Omron CX-Programmer project NewProject (CX-Programmer 9.61)

# PLC NewPLC1: CJ1M CPU21
I/O table (CPU CJ1M-CPU21): rack 0 slot 0 CJ1W-ID211; rack 0 slot 1 CJ1W-OC211; rack 0 slot 2 CJ1W-MAD42

## Global symbols (name address type ; comment)
0.01 BOOL  ; START
1.00 BOOL  ; ON
1.01 BOOL  ; GERAK1
1.02 BOOL  ; GERAK2
1.03 BOOL  ; GERAK3
1.04 BOOL  ; PENGISIAN
2005 CHANNEL  ; LEVEL
T0004 BOOL  ; COUNTER

## Program NewProgram1 (cyclic task 0)

### Section Section1

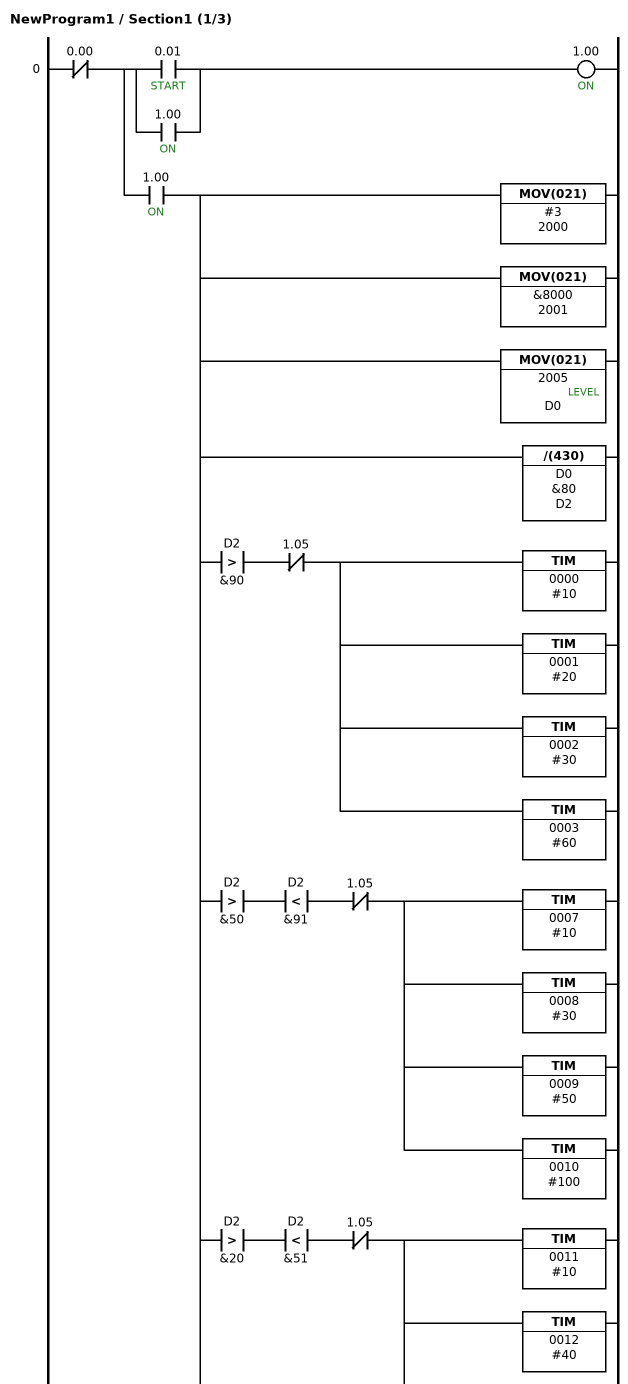

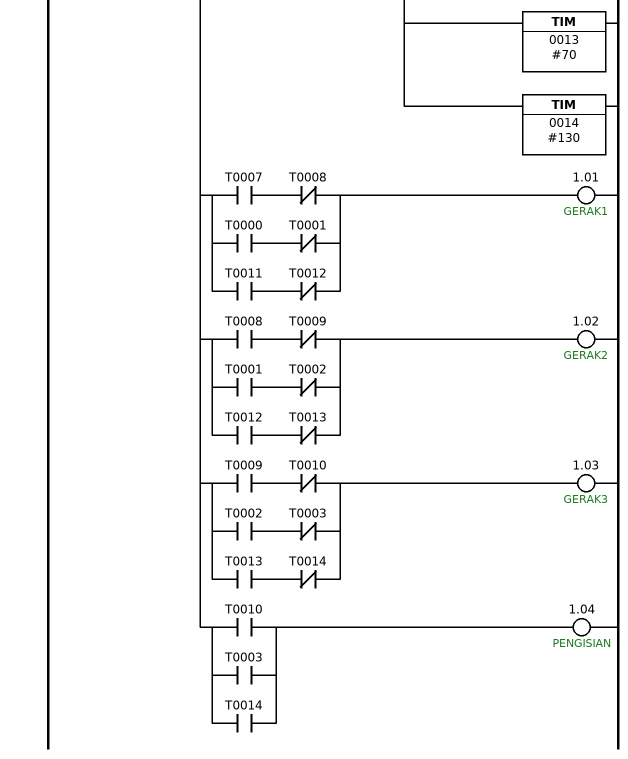
; rung 0
LDNOT 0.00
OUT TR0
LD 0.01  ; START
OR 1.00  ; ON
ANDLD
OUT 1.00  ; ON
LD TR0
AND 1.00  ; ON
OUT TR0
MOV(021) #3 2000
MOV(021) &8000 2001
MOV(021) 2005 D0  ; LEVEL
/(430) D0 &80 D2
AND>(320) D2 &90
ANDNOT 1.05
TIM 0000 #10
TIM 0001 #20
TIM 0002 #30
TIM 0003 #60
LD TR0
AND>(320) D2 &50
AND<(310) D2 &91
ANDNOT 1.05
TIM 0007 #10
TIM 0008 #30
TIM 0009 #50
TIM 0010 #100
LD TR0
AND>(320) D2 &20
AND<(310) D2 &51
ANDNOT 1.05
TIM 0011 #10
TIM 0012 #40
TIM 0013 #70
TIM 0014 #130
LD TR0
LD T0007
ANDNOT T0008
LD T0000
ANDNOT T0001
ORLD
LD T0011
ANDNOT T0012
ORLD
ANDLD
OUT 1.01  ; GERAK1
LD TR0
LD T0008
ANDNOT T0009
LD T0001
ANDNOT T0002
ORLD
LD T0012
ANDNOT T0013
ORLD
ANDLD
OUT 1.02  ; GERAK2
LD TR0
LD T0009
ANDNOT T0010
LD T0002
ANDNOT T0003
ORLD
LD T0013
ANDNOT T0014
ORLD
ANDLD
OUT 1.03  ; GERAK3
LD TR0
LD T0010
OR T0003
OR T0014
ANDLD
OUT 1.04  ; PENGISIAN

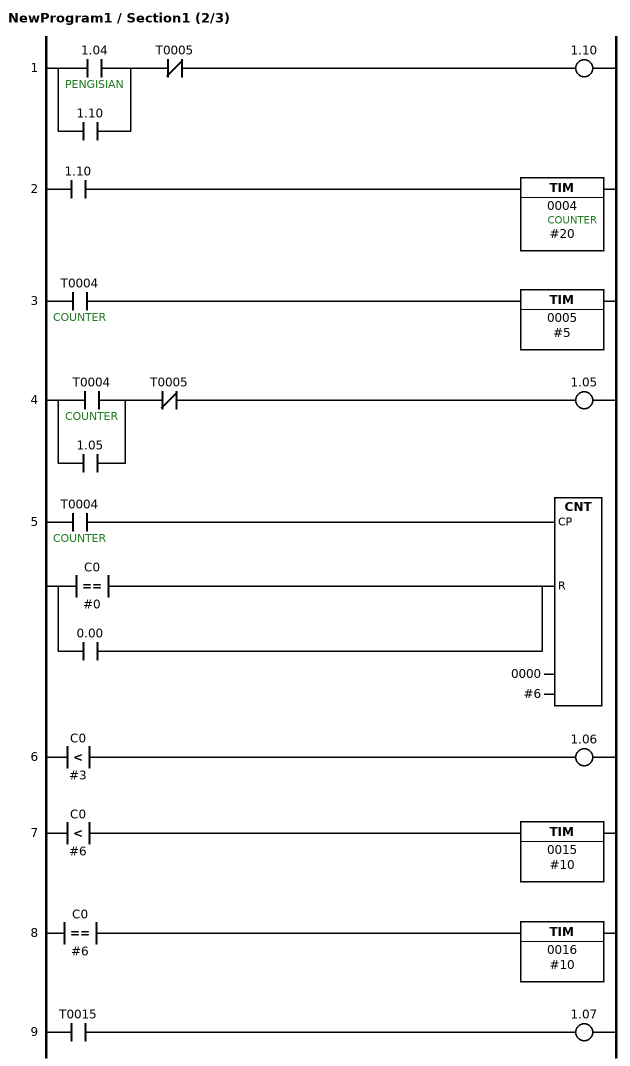
; rung 1
LD 1.04  ; PENGISIAN
OR 1.10
ANDNOT T0005
OUT 1.10
; rung 2
LD 1.10
TIM 0004 #20  ; COUNTER
; rung 3
LD T0004  ; COUNTER
TIM 0005 #5
; rung 4
LD T0004  ; COUNTER
OR 1.05
ANDNOT T0005
OUT 1.05
; rung 5
LD T0004  ; COUNTER
LD=(300) C0 #0
OR 0.00
CNT 0000 #6
; rung 6
LD<(310) C0 #3
OUT 1.06
; rung 7
LD<(310) C0 #6
TIM 0015 #10
; rung 8
LD=(300) C0 #6
TIM 0016 #10
; rung 9
LD T0015
OUT 1.07

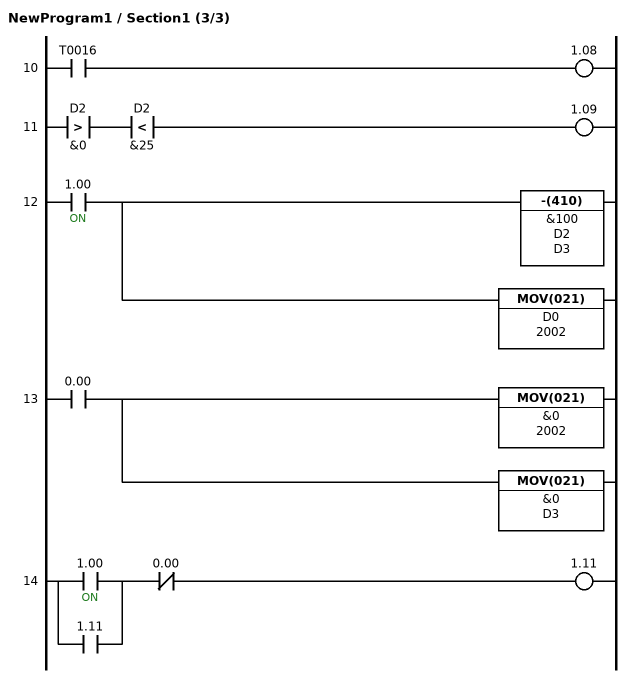
; rung 10
LD T0016
OUT 1.08
; rung 11
LD>(320) D2 &0
AND<(310) D2 &25
OUT 1.09
; rung 12
LD 1.00  ; ON
-(410) &100 D2 D3
MOV(021) D0 2002
; rung 13
LD 0.00
MOV(021) &0 2002
MOV(021) &0 D3
; rung 14
LD 1.00  ; ON
OR 1.11
ANDNOT 0.00
OUT 1.11

### Section END
; rung 0
END(001)